(* Schneider Machine Expert - Basic project Altivar32 (2), file version 1.2.0.0 *)

HARDWARE
  Cpu 0: TM221ME16T/G
  EthernetConfiguration: NetworkName=M221, IpAllocationMode=FixedAddress, IpAddress=10.10.1.135, SubnetMask=255.0.0.0
  SerialLineConfiguration: Baud=Baud19200, Parity=ParityEven, DataBits=DataBits8, StopBits=StopBits1, PhysicalMedium=PhysicalMediumRs485, TransmissionMode=TransmissionModeModbusRtu, SlaveId=1, Addressing=MasterAddressing
  MastTask: UsePeriodScanMode=false, PeriodScan=100
  FastTask: Period=255
  CpuBehavior: StartingMode=StartInRun, AutoSaveRamOnEeprom=true, WatchdogPeriod=250

SYMBOLS  (address, symbol, comment, settings)
  %S5       SB_TB100MS  "Time base of 100 ms generated by an internal clock"
  %MW0      SET_CMD
  %MW1      SET_FREQ
  %MW2      SET_ACC
  %MW3      SET_DEC
  %MW4      SET_HSP
  %MW5      SET_LSP
  %MW10     READ_ETA
  %MW11     READ_SPEED
  %MW12     READ_FREQ
  %WRITE_VAR0   [Link(Id=Link, VisibleName=Link, CompiledType=Word, OfflineAccessRight=ReadWrite, OnlineAccessRight=ReadWrite, IsRuntime=true, Value(FBComLinkParameterEnums=SerialLine1), DefaultValue(FBComLinkParameterEnums=SerialLine1)), RemoteDeviceId(Id=RemoteDeviceId, VisibleName=Id, CompiledType=Word, OfflineAccessRight=ReadWrite, OnlineAccessRight=ReadWrite, IsRuntime=true, Value(int=1), DefaultValue(int=1),]
  %WRITE_VAR1   [Link(Id=Link, VisibleName=Link, CompiledType=Word, OfflineAccessRight=ReadWrite, OnlineAccessRight=ReadWrite, IsRuntime=true, Value(FBComLinkParameterEnums=SerialLine1), DefaultValue(FBComLinkParameterEnums=SerialLine1)), RemoteDeviceId(Id=RemoteDeviceId, VisibleName=Id, CompiledType=Word, OfflineAccessRight=ReadWrite, OnlineAccessRight=ReadWrite, IsRuntime=true, Value(int=1), DefaultValue(int=1),]
  %READ_VAR0   [Link(Id=Link, VisibleName=Link, CompiledType=Word, OfflineAccessRight=ReadWrite, OnlineAccessRight=ReadWrite, IsRuntime=true, Value(FBComLinkParameterEnums=SerialLine1), DefaultValue(FBComLinkParameterEnums=SerialLine1)), RemoteDeviceId(Id=RemoteDeviceId, VisibleName=Id, CompiledType=Word, OfflineAccessRight=ReadWrite, OnlineAccessRight=ReadWrite, IsRuntime=true, Value(int=1), DefaultValue(int=1),]

POU Nouveau POU
  (* SectionNumber=1, IsGrafcet=false *)

// Rung 0
  BLK %WRITE_VAR0
  LD %S5                  (* SB_TB100MS *)
  AND( %READ_VAR0.DONE
  ORN %M1
  )
  Execute
  OUT_BLK
  LD Done
  ST %M1
  END_BLK
  // as ST:
  //   %WRITE_VAR0(EXECUTE := SB_TB100MS AND (%READ_VAR0.DONE OR NOT %M1));
  //   %M1 := %WRITE_VAR0.Done;
  (* the ladder stored for this rung does not match its IL; not drawn *)

// Rung 1
  BLK %WRITE_VAR1
  LD %WRITE_VAR0.DONE
  Execute
  END_BLK
  // as ST:
  //   %WRITE_VAR1(EXECUTE := %WRITE_VAR0.DONE);
  (* the ladder stored for this rung does not match its IL; not drawn *)

// Rung 2
  BLK %READ_VAR0
  LD %WRITE_VAR1.DONE
  Execute
  END_BLK
  // as ST:
  //   %READ_VAR0(EXECUTE := %WRITE_VAR1.DONE);
  (* the ladder stored for this rung does not match its IL; not drawn *)
